// TIA Portal V17 export
// export: Created 2025-08-05T09:35:58.3231078Z, ExportSetting WithDefaults, DisplayName Totally Integrated Automation Portal, DisplayVersion V17, DisplayName TIA Portal Openness, DisplayVersion V17, DisplayName TIA Portal Version Control Interface, DisplayVersion V17, DisplayName SINAMICS Startdrive Advanced, DisplayVersion V17, DisplayName SINAMICS Startdrive G130, G150, S120, S150, SINAMICS MV, S210, DisplayVersion V17, DisplayName SINAMICS Startdrive G110M, G120, G120C, G120D, G120P, G115D, DisplayVersion V17, DisplayName STEP 7 Professional, DisplayVersion V17, DisplayName STEP 7 Safety, DisplayVersion V17, DisplayName WinCC Advanced, DisplayVersion V17
DATA_BLOCK "LaserComm"   // DB295
{ S7_Optimized_Access := 'FALSE' }
VERSION : 0.1
// stored: AutoNumber true, DBAccessibleFromOPCUA true, DBAccessibleFromWebserver true, IsOnlyStoredInLoadMemory false, IsWriteProtectedInAS false
   VAR RETAIN
      "Version" : DInt;
      LDD_Array_Size : DInt;
      Instance : Array[0.."LASERCOMM_NUMBER_OF_LASERS"] of "LaserComm_Instance";
      "this CU" : "typeCaCgFg";
      fg_ControlGeneral { S7_SetPoint := 'True'} : "typeFgControlGeneral";
   END_VAR
BEGIN
END_DATA_BLOCK
